PROGRAM MAIN
VAR
END_VAR

END_PROGRAM

(* stored: Version 1.1.0.1
   POU MAIN: Id {a7dc45c9-34af-4368-8ac0-2e764952b308} *)
